// TIA Portal V19 export
TYPE "LEXCHANGETRAY_typeVfd_par"
// stored: Access Published
   STRUCT
      dec : Real;   // Deceleration Time (seconds)
      acc : Real;   // Acceleration Time (seconds)
      fastDec : Real;   // Fast Stop Deceleration Time (seconds)
      highVel : Real;   // Maximum Operating Speed
      lowVel : Real;   // Minimum Operating Speed
      parentReferenceDesignator : WString[128];
      hwID : HW_IO;   // Hardware Identification Number
      direction : DInt := 1;   // Rotation Direction (1:Clockwise, -1:Counter-clockwise)
   END_STRUCT;
END_TYPE
